(* PLC project Unnamed, Unknown Unnamed 1 *)
(* stored: creationDateTime 2026-07-08T19:42:46, modificationDateTime 2026-07-08T19:42:46 *)

PROGRAM main
  VAR
    output AT %MW0 : INT := 0;
  END_VAR

            output := output + 1;
          
END_PROGRAM

CONFIGURATION Config0
  RESOURCE Res0 ON PLC
    TASK task0(INTERVAL := T#200ms, PRIORITY := 0);
    PROGRAM instance0 WITH task0 : main;
  END_RESOURCE
END_CONFIGURATION
